{attribute addProperty BoxType "EJ7211-0011-0026"}
{attribute addProperty Id "StatuswordAT %I*UINT162"}
{attribute addProperty CRC "1405865676"}
{attribute addProperty SizeInBites "16"}
{attribute addProperty SizeInBytes "2"}
TYPE DS402_Statusword_53CBCECC :
STRUCT
	{attribute addProperty Name "Statusword"}
	Statusword AT %I* : UINT;
END_STRUCT
END_TYPE

(* stored: Version 1.2.0.0, ProductVersion 3.1.4024.9
   DUT DS402_Statusword_53CBCECC: Id {54951e6c-5084-41f2-9a9d-9a497d0854c7} *)
